PROGRAM MAIN
VAR
END_VAR

END_PROGRAM

(* stored: Version 1.1.0.1
   POU MAIN: Id {096234e0-df2d-465f-9000-551e434a4cd4} *)
